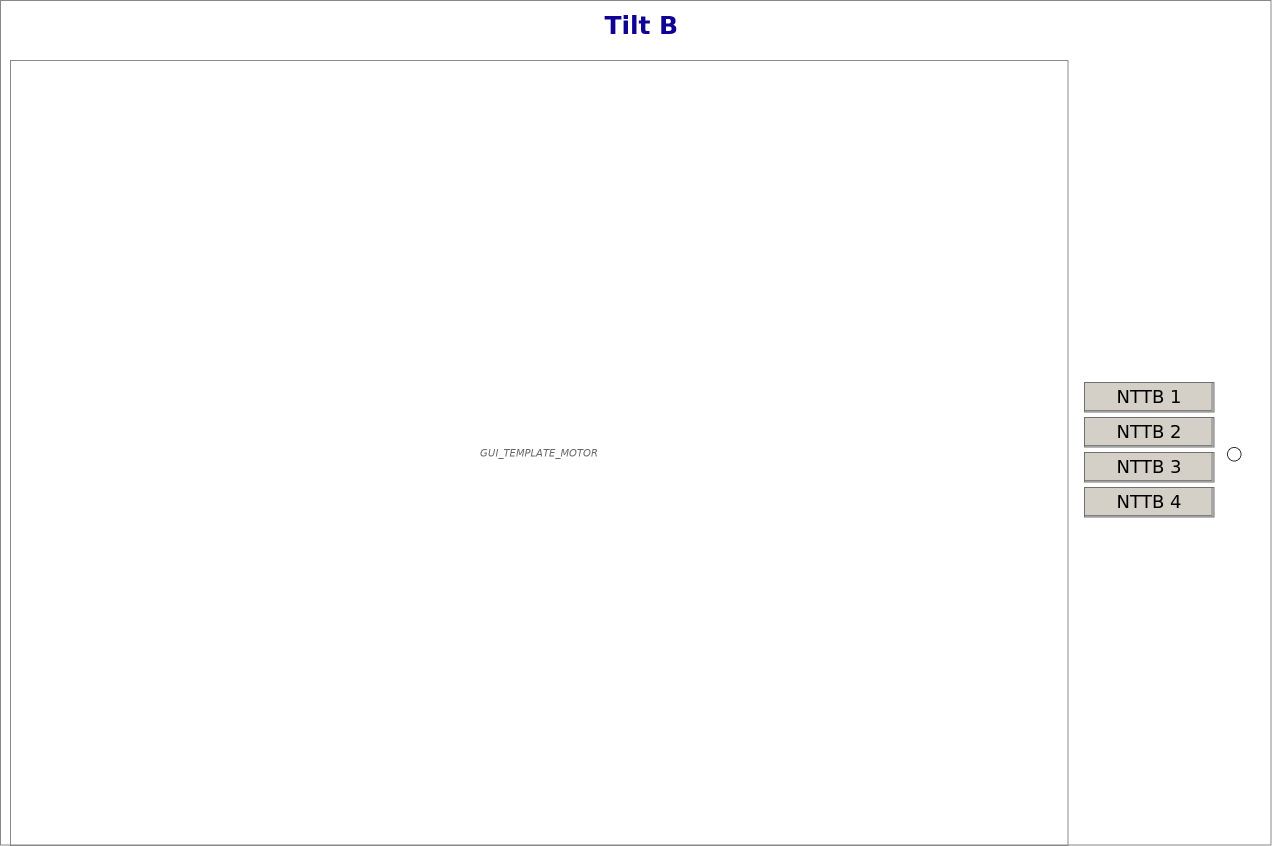
VISUALIZATION VISU_HMI_TILT_B  // 1272x846
    Label (542,10 199x30), "Tilt B"
    Group (10,60 1262x786)
        Frame (0,0 1058x786)
            shows GUI_TEMPLATE_MOTOR(m_Instance := MAIN.nott_ics.TipTilt.ptrTiltActuatorsB[MAIN.nott_ics.TipTilt.guiTiltActuatorsBIndex]^)
        Group (1074,322 188x142)
            RadioButton (141,2 47x140), variable: MAIN.nott_ics.TipTilt.guiTiltActuatorsBIndex-1
                Areas[0]: Text=Radiobutton
                Areas[1]: Text=Radiobutton
            Button (0,0 130x30), "NTTB 1"
                OnMouseClick: execute { MAIN.nott_ics.TipTilt.guiTiltActuatorsBIndex := 1; }
            Button (0,35 130x30), "NTTB 2"
                OnMouseClick: execute { MAIN.nott_ics.TipTilt.guiTiltActuatorsBIndex := 2; }
            Button (0,70 130x30), "NTTB 3"
                OnMouseClick: execute { MAIN.nott_ics.TipTilt.guiTiltActuatorsBIndex := 3; }
            Button (0,105 130x30), "NTTB 4"
                OnMouseClick: execute { MAIN.nott_ics.TipTilt.guiTiltActuatorsBIndex := 4; }
END_VISUALIZATION

(* stored: Version 1.1.0.1, ProductVersion 3.1.4024.14
   Visu VISU_HMI_TILT_B: Id {37561035-cf46-4169-82ee-beddd6e9f3fd} *)
